// Mitsubishi GX Works2 project: 서보제어   PLC: Q03UD

PROGRAM MAIN
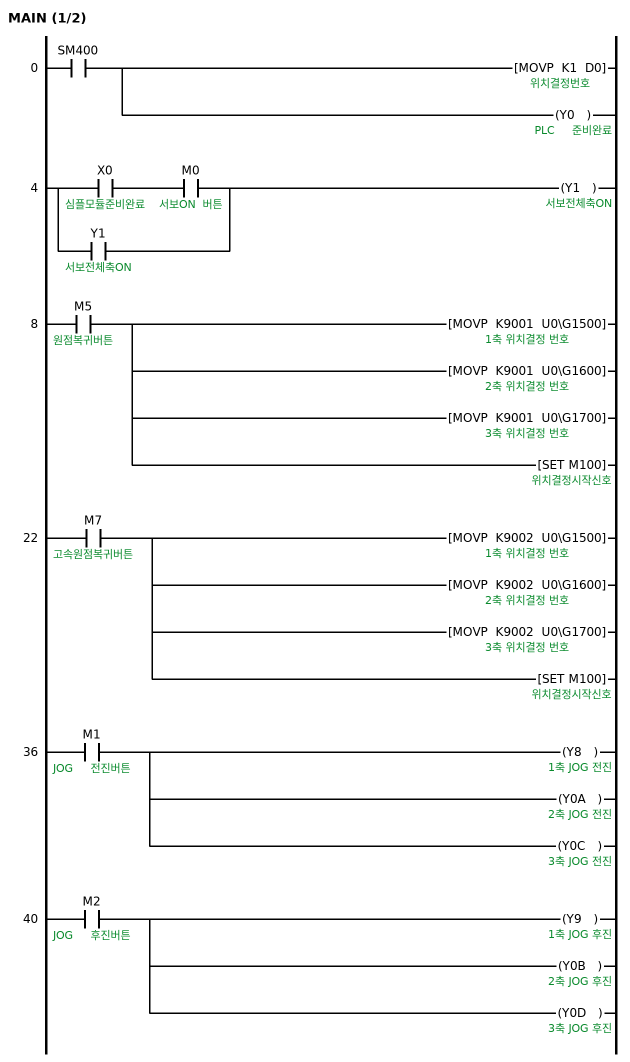
0     LD      SM400
      MOVP    K1 D0  ; 위치결정번호
      OUT     Y0  ; PLC     준비완료
4     LD      X0  ; 심플모듈준비완료
      AND     M0  ; 서보ON  버튼
      OR      Y1  ; 서보전체축ON
      OUT     Y1  ; 서보전체축ON
8     LD      M5  ; 원점복귀버튼
      MOVP    K9001 U0\G1500  ; 1축 위치결정 번호
      MOVP    K9001 U0\G1600  ; 2축 위치결정 번호
      MOVP    K9001 U0\G1700  ; 3축 위치결정 번호
      SET     M100  ; 위치결정시작신호
22    LD      M7  ; 고속원점복귀버튼
      MOVP    K9002 U0\G1500
      MOVP    K9002 U0\G1600
      MOVP    K9002 U0\G1700
      SET     M100  ; 위치결정시작신호
36    LD      M1  ; JOG     전진버튼
      OUT     Y8  ; 1축 JOG 전진
      OUT     Y0A  ; 2축 JOG 전진
      OUT     Y0C  ; 3축 JOG 전진
40    LD      M2  ; JOG     후진버튼
      OUT     Y9  ; 1축 JOG 후진
      OUT     Y0B  ; 2축 JOG 후진
      OUT     Y0D  ; 3축 JOG 후진
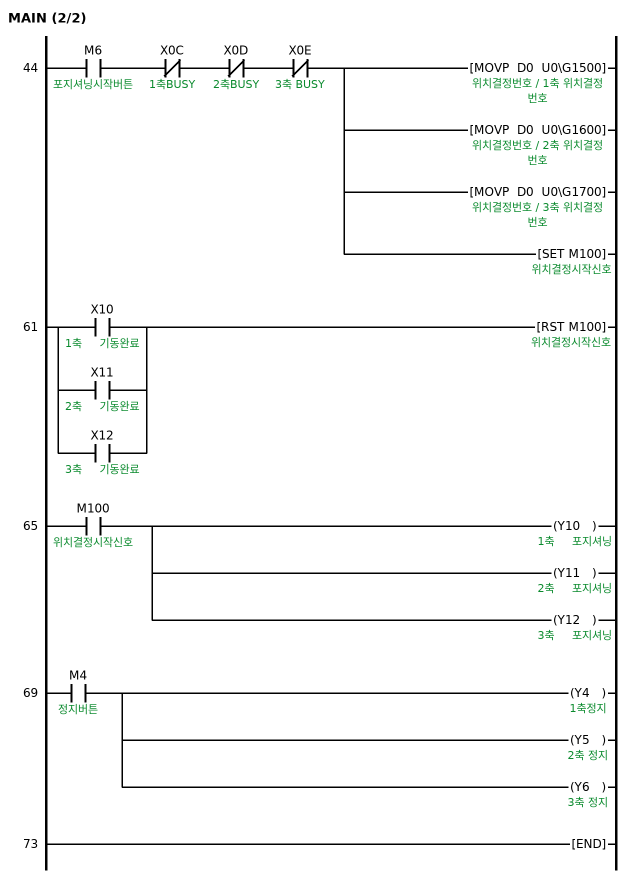
44    LD      M6  ; 포지셔닝시작버튼
      ANI     X0C  ; 1축BUSY
      ANI     X0D  ; 2축BUSY
      ANI     X0E  ; 3축 BUSY
      MOVP    D0 U0\G1500
      MOVP    D0 U0\G1600
      MOVP    D0 U0\G1700
      SET     M100  ; 위치결정시작신호
61    LD      X10  ; 1축     기동완료
      OR      X11  ; 2축     기동완료
      OR      X12  ; 3축     기동완료
      RST     M100  ; 위치결정시작신호
65    LD      M100  ; 위치결정시작신호
      OUT     Y10  ; 1축     포지셔닝
      OUT     Y11  ; 2축     포지셔닝
      OUT     Y12  ; 3축     포지셔닝
69    LD      M4  ; 정지버튼
      OUT     Y4  ; 1축정지
      OUT     Y5  ; 2축 정지
      OUT     Y6  ; 3축 정지
73    END
END_PROGRAM

// device comments not shown above
M3  ; 리셋버튼
